(* Logix 5000 project; controller PLCbox vendor 1 type 14 code 149 rev 30.11; software revision 30.01 *)

TASK MainTask (continuous, watchdog 500 ms) : MainProgram, TestProgram, ExternalHardware, Riser, RPiEdgeIgnition, DellEdgeIgnition
TASK Projects (periodic, rate 10 ms, priority 10, watchdog 500 ms) : StreetLightSystem, PLC_Projects
TASK ST_Routines (periodic, rate 10 ms, priority 10, watchdog 500 ms) : ST_Practice
TASK Task100msec (periodic, rate 100 ms, priority 2, watchdog 500 ms) : MainProgram2
TASK Tutorials (periodic, rate 10 ms, priority 10, watchdog 500 ms) : Mathematical, InterviewPractice, CognexJobChange, Challenges_Projects, TankFillingChallenge, FTViewTutorial, Advanced, PowerFlex525Mastery, FIFOinstruction, JumpTest, DataTypes, PF525Control

MODULES
   Local : vendor 1 type 14 code 149 (Compact 0, rev 30.11)
      Discrete_IO : Embedded (Compact 1, rev 3.1, Output RPI 20 ms)
      CLX_PLC : 1756-EN2T (Ethernet 192.168.1.30, rev 5.28)
         CLX_MainPLC : vendor 1 type 14 code 54 (ICP 0, rev 20.4, $4ae8c327$ RPI 20 ms)
      PF1 : PowerFlex 525-EENET (Ethernet 192.168.1.7, rev 5.2, Output RPI 20 ms)
      Stratix1 : vendor 1 type 12 code 231 (Ethernet 192.168.1.10, rev 8.1, Output RPI 1000 ms)
      VladCognex : vendor 678 type 100 code 265 (Ethernet 192.168.1.15, rev 4.10, Output RPI 20 ms)
      Stratix2 : vendor 1 type 12 code 189 (Ethernet 192.168.1.12, rev 12.1, Output RPI 1000 ms)
      PointIORack1 : 1734-AENT (Ethernet 192.168.1.9, rev 5.1, Output RPI 20 ms)
         Local_IN2 : 1734-IB8 (PointIO 2, rev 3.1)
         Local_IN1 : 1734-IB8 (PointIO 1, rev 3.1)
         Local_OUT5 : vendor 1 type 7 code 288 (PointIO 5, rev 3.1)
         Local_OUT3 : 1734-OB8E (PointIO 3, rev 3.1)
         Local_IN4 : 1734-OA4 (PointIO 4, rev 3.1)
END_MODULES

TYPE String20 :
STRUCT
   LEN : DINT;
   DATA : SINT[20];
END_STRUCT
END_TYPE

TYPE UDT_BOOLarr :
STRUCT
   BOOLtag : BOOL[32];
END_STRUCT
END_TYPE

TYPE UDT_Output :
STRUCT
   Energize : BOOL;
   Auto : BOOL;
   ManualAvl : BOOL;
   Force : BOOL;
   ForceAvl : BOOL;
   Delay_ON : TIMER;
   Name : String20;
   SetAuto : BOOL;
   SetManual : BOOL;
   ForceON : BOOL;
   ForceOFF : BOOL;
END_STRUCT
END_TYPE

TYPE UDT_PID :
STRUCT
   P : REAL;
   I : REAL;
   D : REAL;
   CV : REAL;
   SP : REAL;
   PV : REAL;
   Auto : BOOL;
   Name : STRING;
END_STRUCT
END_TYPE

TYPE UDT_ProdCons :
STRUCT
   Status : CONNECTION_STATUS;
   Data : DINT[50];
END_STRUCT
END_TYPE

TYPE UDT_Time :
STRUCT
   Year : DINT;
   Month : DINT;
   Day : DINT;
   Hour : DINT;
   Minute : DINT;
   Second : DINT;
   Microsecond : DINT;
END_STRUCT
END_TYPE

TYPE UDT_VFD_PF525 :
STRUCT
   Start_PB : BOOL;
   Stop_PB : BOOL;
   Run : BOOL;
END_STRUCT
END_TYPE

TYPE Varchar40 :
STRUCT
   LEN : DINT;
   DATA : SINT[40];
END_STRUCT
END_TYPE

ADD_ON_INSTRUCTION AOI_BasicCalculation   (* revision 1.0, vendor SolisPLC *)
VAR_INPUT
   Operand_1 : REAL; {required}
   Operand_2 : REAL; {required}
   Operand_3 : REAL; {required}
   Operand_4 : REAL; {required}
END_VAR
VAR_OUTPUT
   Multiplication : REAL; {access Read Only, required}
   Addition : REAL; {access Read Only, required}
END_VAR
VAR
   Mul1 : REAL; {access None}
   Mul2 : REAL; {access None}
   Add1 : REAL; {access None}
   Add2 : REAL; {access None}
END_VAR

ROUTINE Logic   (* ladder *)
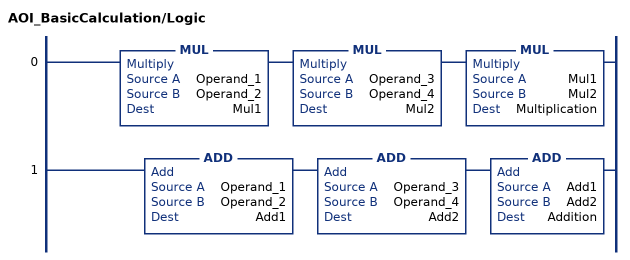
   0: MUL(Operand_1,Operand_2,Mul1)MUL(Operand_3,Operand_4,Mul2)MUL(Mul1,Mul2,Multiplication);
   1: ADD(Operand_1,Operand_2,Add1)ADD(Operand_3,Operand_4,Add2)ADD(Add1,Add2,Addition);
END_ROUTINE
END_ADD_ON_INSTRUCTION

ADD_ON_INSTRUCTION AOI_VFD_PF525   (* revision 1.0, vendor SolisPLC *)
VAR_IN_OUT
   VFD : UDT_VFD_PF525; {required}
END_VAR

ROUTINE Logic   (* structured text *)
   
END_ROUTINE
END_ADD_ON_INSTRUCTION

VAR_GLOBAL   (* controller tags *)
   AnalogInput : REAL[100] := ([0] := 5000.0);
   AnalogScaled : REAL[100] := ([0] := 93.75);
   ArrayOfBOOLs : DINT;
   BNOT_1501 : FBD_BOOLEAN_NOT := (In := 1);
   BOOL_IN_0 : BOOL;
   BOOL_OUT_0 : BOOL;
   BoxCounter : COUNTER := (PRE := 10, ACC := 10, DN := 1);
   Buttons : BOOL[64];
   Buttons2 : UDT_BOOLarr;
   Ch1_Volts : REAL;
   CLX_Cons : UDT_ProdCons := (Status.ConnectionFaulted := 1);
   CMPLX_Prod : UDT_ProdCons := (Status.RunMode := 1, Data[0] := 56789, Data[5] := 674); {produced}
   Command : BOOL[64];
   Condition : BOOL[32];
   Conv1Speed : REAL := 2.0;
   Conv2Speed_Fast : REAL := 3.0;
   Conv2Speed_Slow : REAL := 0.3;
   DINT_Arr1 : DINT[40] := ([0] := 1, [12] := 34534535, [31] := 131231, [34] := 123123);
   DINT_Arr2 : DINT[40] := ([0] := 1, [12] := 34534535, [31] := 131231);
   FaultedT : TIMER := (PRE := 2000, ACC := 860, EN := 1, TT := 1);
   FIFOControl3 : CONTROL := (LEN := 13, POS := 12);
   FIO_B_IN_0 : BOOL;   // Start Button
   FIO_B_IN_1 : BOOL := 1;   // Stop Button
   FIO_B_IN_2 : BOOL;   // System Running
   FIO_B_IN_3 : BOOL;   // Reset Button
   FIO_B_IN_4 : BOOL;
   FIO_B_IN_5 : BOOL;
   FIO_B_OUT_0 : BOOL;   // System Running - Confirmation
   FIO_B_OUT_1 : BOOL := 1;   // System Stopped - Confirmation
   FIO_B_OUT_2 : BOOL;   // System Faulted - Confirmation
   FIO_B_OUT_3 : BOOL := 1;   // Send boxes
   FIO_B_OUT_4 : BOOL := 1;
   FIO_B_OUT_5 : BOOL;
   FIO_B_OUT_6 : BOOL;
   FIO_F_OUT_0 : REAL;
   FIO_F_OUT_1 : REAL;
   FORDINT : DINT[30];
   FORDINT2 : DINT[30];
   HeatingSystem : REAL;
   HMI_Int_BOOL : BOOL[64] := ([5] := 1);
        [1]   // Light 1 Status - Yellow
        [2]   // Light 1 Status - Red
        [4]   // Light 2 Status - Yellow
        [5]   // Light 2 Status - Red
        [0]   // Light 1 Status - Green
        [3]   // Light 2 Status - Green
   HMI_Interface_BOOL : BOOL[64];
        [2]   // Light 1 - Red Status ON
        [5]   // Light 2 - Red Status ON
        [0]   // Light 1 - Green Status ON
        [1]   // Light 1 - Yellow Status ON
        [3]   // Light 2 - Green Status ON
        [4]   // Light 2 - Yellow Status ON
   HMI_No_Access : BOOL;
   IN_Loc1 : BOOL[32];
        [1]   // SPARE
        [2]   // SPARE
        [3]   // SPARE
        [4]   // SPARE
        [5]   // SPARE
        [6]   // SPARE
        [0]   // Box Counter P.E. - No Box
        [7]   // SPARE
   IN_Loc1_DB_OFF : BOOL[32];
   IN_Loc1_DB_ON : BOOL[32];
   IN_Loc1_Index : DINT := 7;
   IN_Loc1_T_OFF : TIMER[16] := ([0].PRE := 500, [0].ACC := 500);
   IN_Loc1_T_ON : TIMER[16] := ([0].PRE := 500);
   index : DINT := 50;
   JobData : SINT[32] := ([0] := 16, [2] := 70, [3] := 105, [4] := 114, [5] := 115, [6] := 116, [7] := 74, [8] := 111, [9] := 98, [10] := 84, [11] := 101, [12] := 115, [13] := 116, [14] := 46, [15] := 106, [16] := 111, [17] := 98);
   Light1_Complete_ONS : BOOL;
   Light1_Green : BOOL;
   Light1_Green_T : TIMER := (PRE := 10000);
   Light1_Red : BOOL;
   Light1_Reset : BOOL;
   Light1_Yellow : BOOL;
   Light1_Yellow_T : TIMER := (PRE := 3000);
   Light2_Complete_ONS : BOOL;
   Light2_Green : BOOL;
   Light2_Green_T : TIMER := (PRE := 10000);
   Light2_Red : BOOL;
   Light2_Reset : BOOL;
   Light2_Yellow : BOOL;
   Light2_Yellow_T : TIMER := (PRE := 3000);
   LightSystem_FLT : BOOL[64] := ([3] := 1);
        [1]   // FLT[1] - Light 1 - Yellow Light Faulted
        [0]   // FLT[0] - Light 1 - Green Light Faulted
   LightSystemFaulted : BOOL := 1;
   Local2IData : DINT := 53;
   Local3OData : DINT := 32;
   Local_IN_D : BOOL[256] := ([0] := 1, [2] := 1, [4] := 1, [5] := 1);
        [1]   // Light 1 - Yellow Light Corfirmed ON
        [0]   // Light 1 - Green Light Corfirmed ON
        [4]   // Light 2 - Yellow Light Corfirmed ON
        [2]   // Light 1 - Red Light Corfirmed ON
        [3]   // Light 2 - Green Light Corfirmed ON
        [5]   // Light 2 - Red Light Corfirmed ON
   Local_OUT_D : BOOL[256] := ([2] := 1);
        [0]   // Light 1 - Green Light Turn ON
        [2]   // Light 1 - Red Light Turn ON
        [3]   // Light 2 - Green Light Turn ON
        [1]   // Light 1 - Yellow Light Turn ON
        [5]   // Light 2 - Red Light Turn ON
        [4]   // Light 2 - Yellow Light Turn ON
   LocalOut : DINT[20] := ([2] := 548);
   LogicTag : BOOL[64] := ([12] := 1, [15] := 1);
   LoopDINT : DINT[30];
   LoopDINT2 : DINT[30];
   NewProductID : DINT := 1017;
   OUT_Loc1 : BOOL[32] := ([0] := 1);
   PID1 : PID := (CTL := 33920, INI := 1, DVNA := 1, PVHA := 1, SP := 200.0, KP := 1.0, KI := 0.1, KD := 0.1, MAXS := 1000.0, SO := 20.000076, MAXO := 100.0, UPD := 0.05, PV := 200.00174, ERR := -0.001739502, OUT := 20.000076, MAXI := 1000.0, MAXCV := 1000.0, MAXTIE := 100.0, DATA[0] := 20.00025, DATA[1] := -320.00278, DATA[2] := 200.00174, DATA[3] := -0.001739502, DATA[4] := 200.0, DATA[5] := 0.1, DATA[6] := 1.0, DATA[7] := 0.90000004, DATA[8] := 1.0, DATA[9] := 0.1, DATA[10] := 0.1, DATA[11] := 1.0, DATA[12] := 0.1, DATA[13] := 0.1, DATA[15] := 10.0, DATA[16] := 1.0);
   PID1_CV : REAL := 200.00076;
   PID1_PV : REAL := 200.00174;
   PID1_T : TIMER := (PRE := 50, ACC := 40, EN := 1, TT := 1);
   PID1_TB : REAL;
   PID_Analog_In : REAL[20];
   PID_Tutorial : PID := (CTL := 34432, INI := 1, DVNA := 1, DVPA := 1, PVHA := 1, SP := 100.0, KP := 5.0, KI := 5.0, KD := 5.0, MAXS := 1000.0, SO := 1.999996, MAXO := 100.0, UPD := 0.05, PV := 100.0, OUT := 1.999996, MAXI := 1000.0, MAXCV := 1000.0, MAXTIE := 100.0, DATA[0] := 1.9999565, DATA[1] := -160.00005, DATA[2] := 100.0, DATA[4] := 100.0, DATA[5] := 0.1, DATA[6] := 1.0, DATA[7] := 5.8, DATA[8] := 5.0, DATA[9] := 5.0, DATA[10] := 5.0, DATA[11] := 5.0, DATA[12] := 5.0, DATA[13] := 5.0, DATA[15] := 10.0, DATA[16] := 1.0);
   PLCTime : UDT_Time := (Year := 2020, Month := 4, Day := 20, Hour := 14, Minute := 9, Second := 30, Microsecond := 102344);
   Proj1_INT : INT[4] := ([0] := 16);
        [0].1   // System Faulted
        [0].2   // Enable Conveyor 1
        [0].3   // Enable Conveyor 2
        [0].4   // Conveyor 2 - HIGH SPEED
   RiserBOOL : BOOL[64];
        [7]   // Riser - Stop PB
        [8]   // Riser - Critical Fault
        [0]   // Riser - Cotnrol Valve OPEN
        [9]   // Riser - Fault Reset PB
        [5]   // Riser - Running Condition
        [4]   // Riser ALARM 004 - Pressure High High
        [3]   // Riser ALARM 003 - Pressure High
        [6]   // Riser - Start PB
        [2]   // Riser ALARM 002 - Pressure Low
        [1]   // Riser ALARM 001 - Pressure Low Low
   RiserREAL : REAL[20] := ([0] := 55.0, [1] := 20.0, [2] := 5.0, [3] := 124.80001, [4] := 140.40001, [5] := 140.0, [6] := 156.00002, [7] := 124.80001, [8] := 140.40001, [9] := 4.0, [10] := 4.5);
        [1]   // Riser - Pressure Limit Low Low[PSI]
        [2]   // Riser - Pressure Limit Low [PSI]
        [0]   // Riser - Current Pressure Reading [PSI]
        [6]   // Riser - DR 9 Pipe Pressure Rating [PSI]
        [5]   // Riser - Current Temperature Reading [deg F]
        [4]   // Riser - Pressure Limit High High [PSI]
        [3]   // Riser - Pressure Limit High [PSI]
        [8]   // Riser - Pressure Limit High High [PSI]
        [7]   // Riser - Pressure Limit High [PSI]
   SCLA_10 : SCALE := (In := 5000.0, InRawMax := 16000.0, InEUMax := 300.0, Out := 93.75);
   SCLA_11 : SCALE;
   SCLA_12 : SCALE;
   SetJob : MESSAGE;
        MessageParameters(ServiceCode := 16#0010, LocalElement := JobData[0], ...)
   SolisBOOL : BOOL[64] := ([2] := 1, [3] := 1, [4] := 1, [5] := 1, [7] := 1, [8] := 1, [9] := 1, [10] := 1, [11] := 1, [12] := 1, [13] := 1);
   SolisDINT : DINT[20] := ([2] := 42, [3] := 234, [5] := 234, [6] := 33, [7] := 234, [8] := 234, [9] := 23, [10] := 24, [11] := 42, [12] := 234, [13] := 423, [15] := 42);
   SolisREAL : REAL[20];
   SsytemStopped : BOOL := 1;
   StatusInt : DINT := 2;
   System_Timer : TIMER[100] := ([0].PRE := 10000, [0].ACC := 783, [0].EN := 1, [0].TT := 1);
   SystemFaultReset : BOOL;
   tagToPi : DINT := 119;
   TempSensor : REAL;
   TIC_1501 : PID_ENHANCED := (PVEUMax := 100.0, SPHLimit := 100.0, RatioProg := 1.0, RatioOper := 1.0, RatioHLimit := 1.0, RatioLLimit := 1.0, CVEUMax := 100.0, CVHLimit := 100.0, PVEDerivative := 1, RTSTime := 1);
END_VAR

PROGRAM Advanced   (* main routine _01_Main *)
VAR
   Add : REAL;
   AOI_Basic1 : AOI_BasicCalculation;
   Array1_INT : INT[10] := ([0] := -21846, [1] := -1);
   Array2_DINT : DINT[10] := ([0] := -21846);
   BatchCompletedConfirm : BOOL;
   Data : DINT[50];
   Data2 : DINT[50];
   DestBit : DINT;
   Ingredient1Stp : DINT := 30;
   Ingredient2Stp : DINT := 70;
   Ingredient3Stp : DINT := 99;
   Mult : REAL;
   Op1 : REAL;
   Op2 : REAL;
   Op3 : REAL;
   Op4 : REAL;
   PLCCond : BOOL[32];
        [1]   // Batch Start Button
   PLCCondOut : BOOL[32] := ([1] := 1);
        [8]   // Batch Completed
        [2]   // Ingredient 1 Valve OPEN
        [1]   // Tank Ready for Batch
        [4]   // Enable Stirrer (VFD)
        [5]   // Hops Feeder ENABLE
        [3]   // Ingredient 2 Valve OPEN
        [6]   // Tank Heating System ENABLE
   SeqArr : DINT[10] := ([0] := 1, [1] := 2, [2] := 4, [3] := 12, [4] := 28, [5] := 60, [6] := 124, [7] := 128);
   SeqArr2 : DINT[10] := ([0] := 1, [1] := 2, [2] := 4, [3] := 24, [4] := 48, [5] := 80, [6] := 208, [7] := 256);
   SeqControl : CONTROL := (LEN := 7, POS := 1);
   SeqMask : DINT := 65535;
   SeqOut : DINT := 2;
   SeqSource : DINT;
   SequencePosition : DINT;
   SequenceStart : BOOL;
   SrcBit : DINT;
   TankDelay : TIMER := (PRE := 30000);
   TankLevel : DINT;
   TankTemperature : DINT := 200;
   TankTempStp : DINT := 220;
END_VAR

ROUTINE _01_Main   (* ladder *)
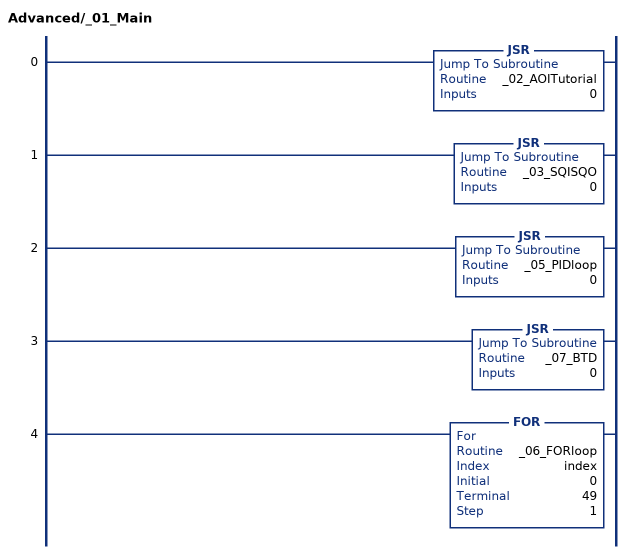
   0: JSR(_02_AOITutorial,0);
   1: JSR(_03_SQISQO,0);
   2: JSR(_05_PIDloop,0);
   3: JSR(_07_BTD,0);
   4: FOR(_06_FORloop,index,0,49,1);
END_ROUTINE

ROUTINE _02_AOITutorial   (* ladder *)
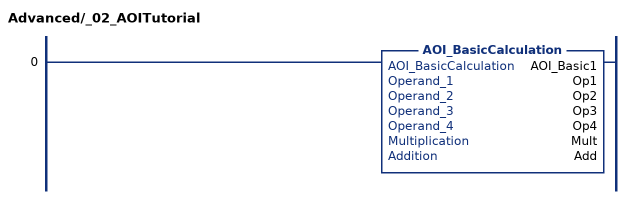
   0: AOI_BasicCalculation(AOI_Basic1,Op1,Op2,Op3,Op4,Mult,Add);
END_ROUTINE

ROUTINE _03_SQISQO   (* ladder *)
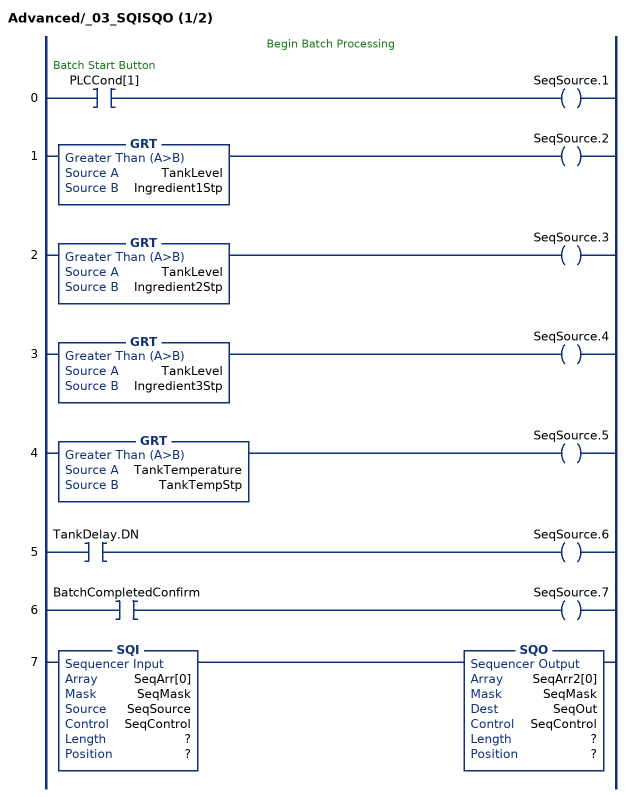
   // Begin Batch Processing
   0: XIC(PLCCond[1])OTE(SeqSource.1);
   1: GRT(TankLevel,Ingredient1Stp)OTE(SeqSource.2);
   2: GRT(TankLevel,Ingredient2Stp)OTE(SeqSource.3);
   3: GRT(TankLevel,Ingredient3Stp)OTE(SeqSource.4);
   4: GRT(TankTemperature,TankTempStp)OTE(SeqSource.5);
   5: XIC(TankDelay.DN)OTE(SeqSource.6);
   6: XIC(BatchCompletedConfirm)OTE(SeqSource.7);
   7: SQI(SeqArr[0],SeqMask,SeqSource,SeqControl,?,?)SQO(SeqArr2[0],SeqMask,SeqOut,SeqControl,?,?);
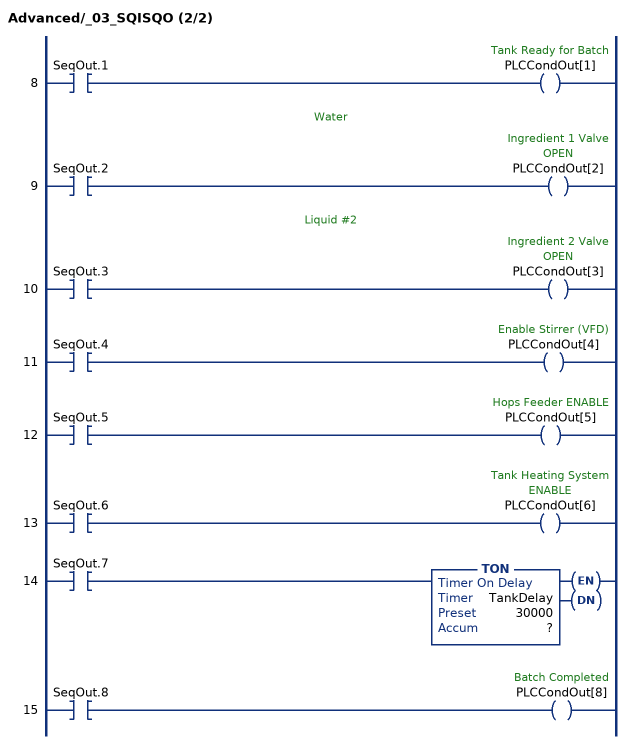
   8: XIC(SeqOut.1)OTE(PLCCondOut[1]);
   // Water
   9: XIC(SeqOut.2)OTE(PLCCondOut[2]);
   // Liquid #2
   10: XIC(SeqOut.3)OTE(PLCCondOut[3]);
   11: XIC(SeqOut.4)OTE(PLCCondOut[4]);
   12: XIC(SeqOut.5)OTE(PLCCondOut[5]);
   13: XIC(SeqOut.6)OTE(PLCCondOut[6]);
   14: XIC(SeqOut.7)TON(TankDelay,?,?);
   15: XIC(SeqOut.8)OTE(PLCCondOut[8]);
END_ROUTINE

ROUTINE _05_PIDloop   (* ladder *)
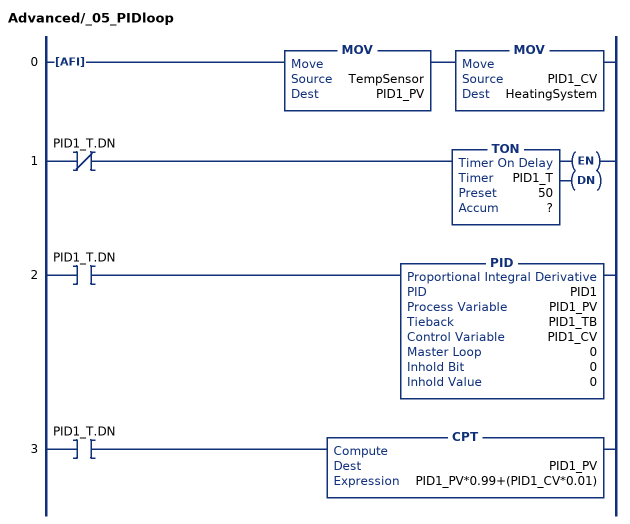
   0: AFI()MOV(TempSensor,PID1_PV)MOV(PID1_CV,HeatingSystem);
   1: XIO(PID1_T.DN)TON(PID1_T,?,?);
   2: XIC(PID1_T.DN)PID(PID1,PID1_PV,PID1_TB,PID1_CV,0,0,0);
   3: XIC(PID1_T.DN)CPT(PID1_PV,PID1_PV*0.99+(PID1_CV*0.01));
END_ROUTINE

ROUTINE _06_FORloop   (* ladder *)
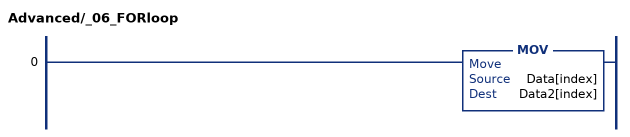
   0: MOV(Data[index],Data2[index]);
END_ROUTINE

ROUTINE _07_BTD   (* ladder *)
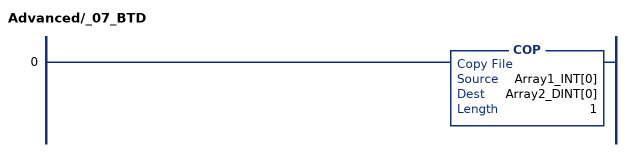
   0: COP(Array1_INT[0],Array2_DINT[0],1);
END_ROUTINE
END_PROGRAM

PROGRAM Challenges_Projects   (* main routine _01_Main *)
VAR
   GREEN_LIGHT_ON : BOOL;
   RED_LIGHT_ON : BOOL;
   RESET_PRESSED : BOOL;
   START_PRESSED : BOOL;
   STOP_PRESSED : BOOL;
   YELLOW_LIGHT_ON : BOOL;
END_VAR

ROUTINE _01_Main   (* ladder *)
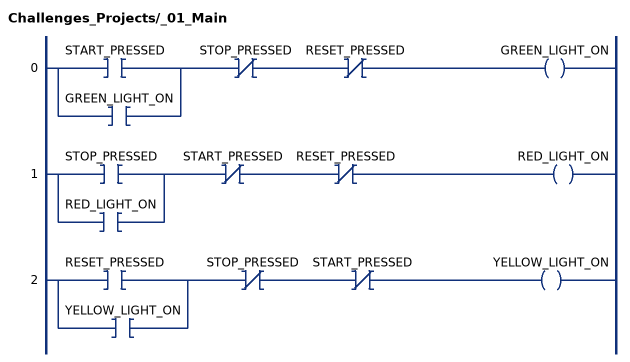
   0: [XIC(START_PRESSED) ,XIC(GREEN_LIGHT_ON) ]XIO(STOP_PRESSED)XIO(RESET_PRESSED)OTE(GREEN_LIGHT_ON);
   1: [XIC(STOP_PRESSED) ,XIC(RED_LIGHT_ON) ]XIO(START_PRESSED)XIO(RESET_PRESSED)OTE(RED_LIGHT_ON);
   2: [XIC(RESET_PRESSED) ,XIC(YELLOW_LIGHT_ON) ]XIO(STOP_PRESSED)XIO(START_PRESSED)OTE(YELLOW_LIGHT_ON);
END_ROUTINE
END_PROGRAM

PROGRAM CognexJobChange   (* main routine Main *)
VAR
   JobIndex : DINT := 1;
   JobName : STRING[10] := ([0] := 'VladsJob.job', [1] := 'FirstJobTest.job', [2] := 'BarcodeRead.job');
   JobSet : BOOL[32];
   JobTrigger : BOOL;
   TriggerONS : BOOL;
   VladsCounter : COUNTER := (ACC := 11, DN := 1);
END_VAR

ROUTINE Main   (* ladder *)
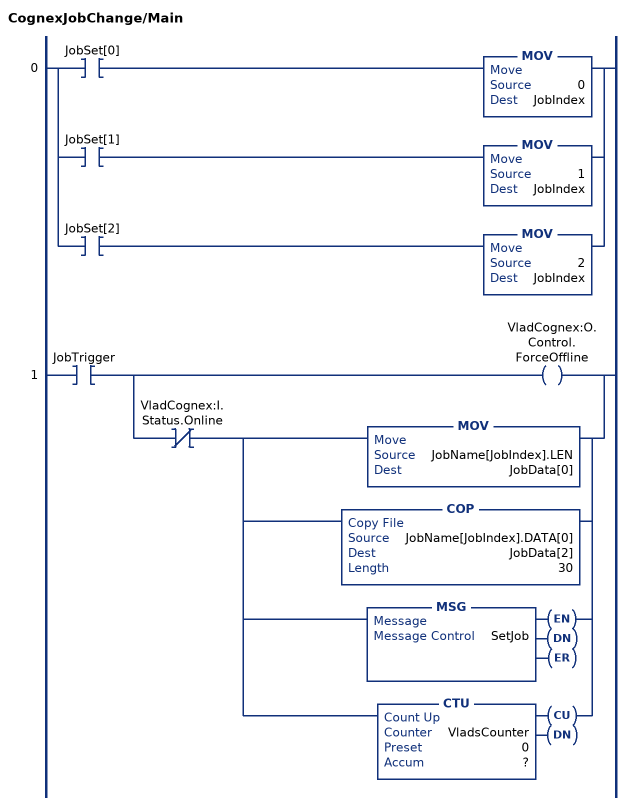
   0: [XIC(JobSet[0]) MOV(0,JobIndex) ,XIC(JobSet[1]) MOV(1,JobIndex) ,XIC(JobSet[2]) MOV(2,JobIndex) ];
   1: XIC(JobTrigger)[OTE(VladCognex:O.Control.ForceOffline) ,XIO(VladCognex:I.Status.Online) [MOV(JobName[JobIndex].LEN,JobData[0]) ,COP(JobName[JobIndex].DATA[0],JobData[2],30) ,MSG(SetJob) ,CTU(VladsCounter,?,?) ] ];
END_ROUTINE
END_PROGRAM

PROGRAM DataTypes   (* main routine _01_Main *)
VAR
   Machine : BOOL := 1;
   Output : DINT := 7;
   Output2 : DINT := 7;
   Output_Buffer1 : DINT := 7;
   Start_Light : BOOL := 1;
   Stop_Light : BOOL := 1;
   Tag1 : BOOL := 1;
   Tag10 : DINT[10] := ([5] := 256);
   Tag2 : INT;
   Tag3 : DINT;
   Tag4 : BOOL[32] := ([2] := 1, [5] := 1, [8] := 1, [11] := 1, [17] := 1);
   Tag5 : DINT;
   Tag6 : BOOL;
   Tag7 : BOOL;
   Tag8 : DINT;
   Tag9 : BOOL;
   ValveOutput : BOOL := 1;
   Warning_Light : BOOL := 1;
END_VAR

ROUTINE _01_Main   (* ladder *)
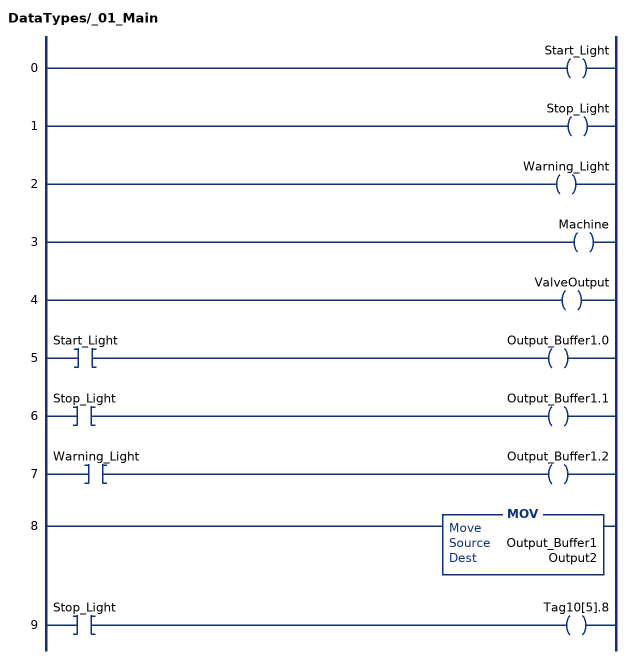
   0: OTE(Start_Light);
   1: OTE(Stop_Light);
   2: OTE(Warning_Light);
   3: OTE(Machine);
   4: OTE(ValveOutput);
   5: XIC(Start_Light)OTE(Output_Buffer1.0);
   6: XIC(Stop_Light)OTE(Output_Buffer1.1);
   7: XIC(Warning_Light)OTE(Output_Buffer1.2);
   8: MOV(Output_Buffer1,Output2);
   9: XIC(Stop_Light)OTE(Tag10[5].8);
END_ROUTINE
END_PROGRAM

PROGRAM DellEdgeIgnition
VAR
   DellIgn_BOOL : BOOL[128];
   DellIgn_DINT : DINT[50] := ([0] := 1);
END_VAR
END_PROGRAM

PROGRAM ExternalHardware   (* main routine _01_Main *)
VAR
   HMI_O_Screeen_Title : String20[100] := ([0] := 'Slot 0 - Local Out.', [1] := 'Main Screen', [2] := 'System Settings', [3] := 'In Q - Motor Starter', [4] := 'Alarm Display');
END_VAR

ROUTINE _01_Main   (* ladder *)
   0 (stored rung type 13): ;
END_ROUTINE
END_PROGRAM

PROGRAM FIFOinstruction   (* main routine FIFOdemo *)
VAR
   BoxCounter2 : COUNTER := (ACC := 1, CU := 1, DN := 1);
   BoxProx2 : BOOL := 1;
   FIFO_Array : DINT[100] := ([0] := 140, [1] := 12910, [2] := 440, [3] := 150, [4] := 150, [5] := 150, [6] := 180, [7] := 300, [8] := 109, [9] := 10, [10] := 130, [11] := 180, [12] := 160, [13] := 240, [14] := 780, [15] := 880, [16] := 300000, [17] := 250, [18] := 150);
   FIFO_Array3 : DINT[100] := ([0] := 1, [1] := 1, [2] := 1, [3] := 1, [4] := 1, [5] := 1, [6] := 1, [7] := 1, [8] := 1, [9] := 1, [10] := 1, [11] := 1);
   FIFO_Unld : DINT := 1;
   FIFOAvg : DINT := 1;
   FIFOControl : CONTROL := (LEN := 20, POS := 19);
   FIFOLength : DINT := 11;
   FIFOSum : DINT := 12;
   SecTime : DINT;
   System_BOOL : BOOL;
   System_BOOL1 : BOOL[64] := ([5] := 1);
   TimerSinceLastBox : TIMER := (PRE := 300000, ACC := 300000, EN := 1, DN := 1);
END_VAR

ROUTINE FIFO_Avg   (* ladder *)
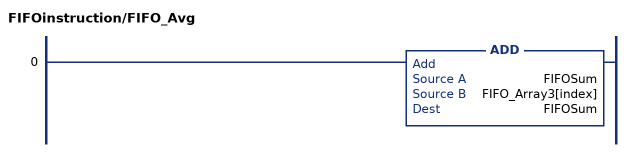
   0: ADD(FIFOSum,FIFO_Array3[index],FIFOSum);
END_ROUTINE

ROUTINE FIFOdemo   (* ladder *)
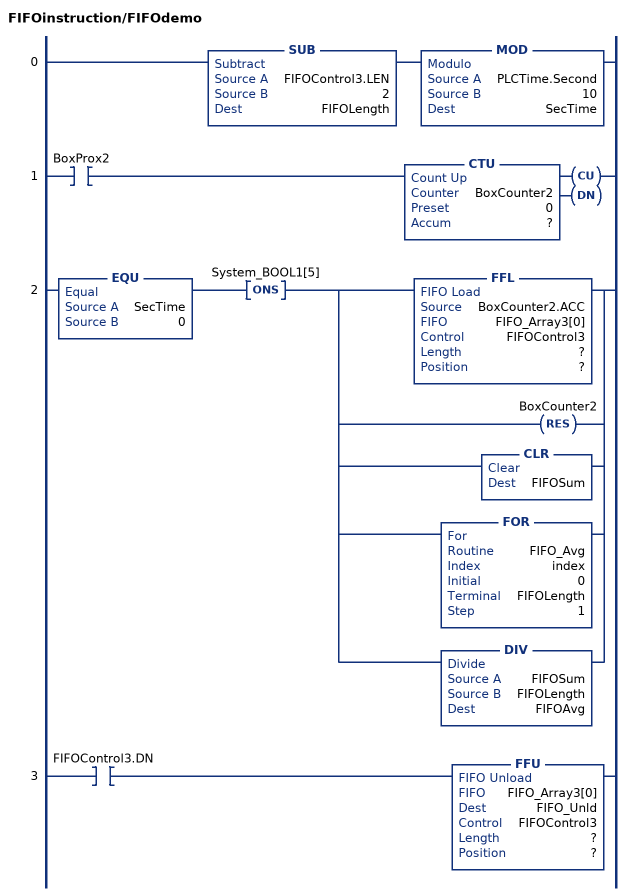
   0: SUB(FIFOControl3.LEN,2,FIFOLength)MOD(PLCTime.Second,10,SecTime);
   1: XIC(BoxProx2)CTU(BoxCounter2,?,?);
   2: EQU(SecTime,0)ONS(System_BOOL1[5])[FFL(BoxCounter2.ACC,FIFO_Array3[0],FIFOControl3,?,?) ,RES(BoxCounter2) ,CLR(FIFOSum) ,FOR(FIFO_Avg,index,0,FIFOLength,1) ,DIV(FIFOSum,FIFOLength,FIFOAvg) ];
   3: XIC(FIFOControl3.DN)FFU(FIFO_Array3[0],FIFO_Unld,FIFOControl3,?,?);
END_ROUTINE
END_PROGRAM

PROGRAM FTViewTutorial   (* main routine _01_Main *)
VAR
   AlarmReset : BOOL;
   HMI_Rotation : TIMER := (PRE := 5000, ACC := 410, EN := 1, TT := 1);
   HMI_Rotation_Enable : BOOL := 1;
   Motor1HL : BOOL;
   Motor1LL : BOOL;
   Motor1Speed : REAL := 60.0;
   Motor1SpeedActual : REAL := 60.0;
   Motor1SpeedSetpoint : REAL := 60.0;
   Motor1Var : REAL := 5.0;
END_VAR

ROUTINE _01_Main   (* ladder *)
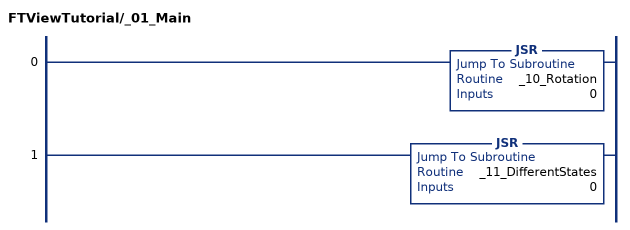
   0: JSR(_10_Rotation,0);
   1: JSR(_11_DifferentStates,0);
END_ROUTINE

ROUTINE _10_Rotation   (* ladder *)
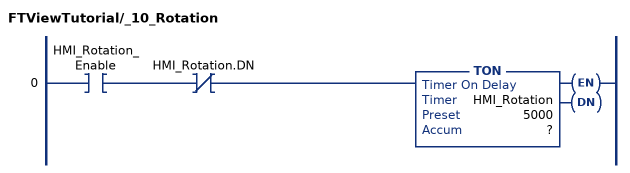
   0: XIC(HMI_Rotation_Enable)XIO(HMI_Rotation.DN)TON(HMI_Rotation,?,?);
END_ROUTINE

ROUTINE _11_DifferentStates   (* ladder *)
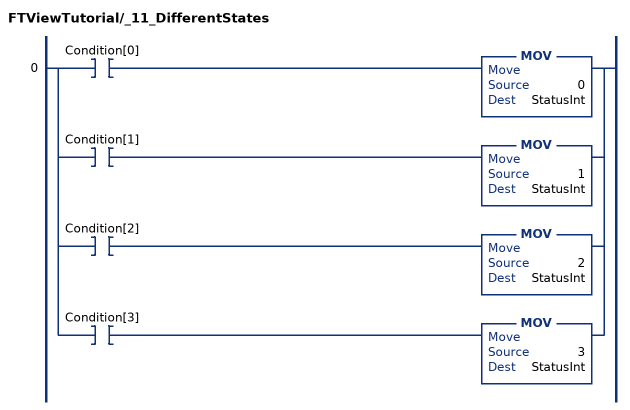
   0: [XIC(Condition[0]) MOV(0,StatusInt) ,XIC(Condition[1]) MOV(1,StatusInt) ,XIC(Condition[2]) MOV(2,StatusInt) ,XIC(Condition[3]) MOV(3,StatusInt) ];
END_ROUTINE
END_PROGRAM

PROGRAM InterviewPractice   (* main routine _01_Main *)
VAR
   AllOn : DINT := 2;
   CurrentRecipe : DINT := 2;
   HMI_RecipeSelected : DINT := 2;
   INT_Motor : BOOL[32];
        [1]   // STOP
        [10]   // MOTOR STARTER
        [0]   // START
        [2]   // MOTOR OVERLOAD / FAULT
   Recipe : DINT[10] := ([0] := 255, [1] := 55);
   RecipeCheck : DINT[10] := ([1] := 55);
   RecipeChk : DINT[10] := ([1] := 55, [2] := 10, [3] := 48);
   RecipeNumber : DINT[10] := ([1] := 55, [2] := 10, [3] := 48);
   SensorValve : DINT := 11;
   test : BOOL := 1;
   ValveBank : BOOL[32];
        [0]   // Valve - Sugar Tank
        [1]   // Valve - Salt Tank
        [2]   // Valve - Spice Tank
        [3]   // Valve - Iodine Tank
   ValveBank2 : BOOL[32] := ([0] := 1, [1] := 1, [2] := 1, [3] := 1, [4] := 1, [5] := 1, [6] := 1);
   ValveBank3 : DINT := 2;
   ValveBits : DINT;
   Valves : DINT := 10;
        .1   // Ingredient Valve - Salt
        .2   // Ingredient Valve - Spices
        .0   // Ingredient Valve - Sugar
        .3   // Ingredient Valve - Malto
   ValvesOK_SystemReady : BOOL;
   ValvesOK_SystemReady2 : BOOL := 1;
   ValvesOpen : DINT := 11;
END_VAR

ROUTINE _01_Main   (* ladder *)
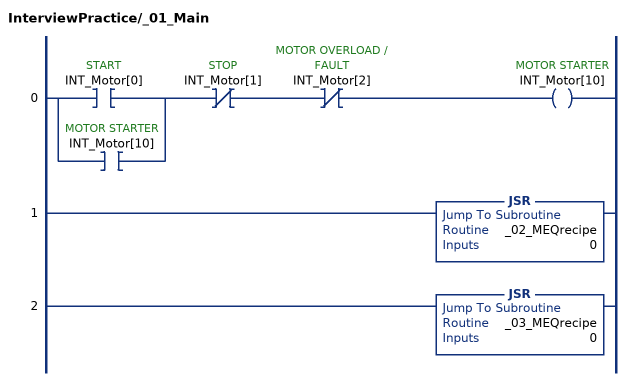
   0: [XIC(INT_Motor[0]) ,XIC(INT_Motor[10]) ]XIO(INT_Motor[1])XIO(INT_Motor[2])OTE(INT_Motor[10]);
   1: JSR(_02_MEQrecipe,0);
   2: JSR(_03_MEQrecipe,0);
END_ROUTINE

ROUTINE _02_MEQrecipe   (* ladder *)
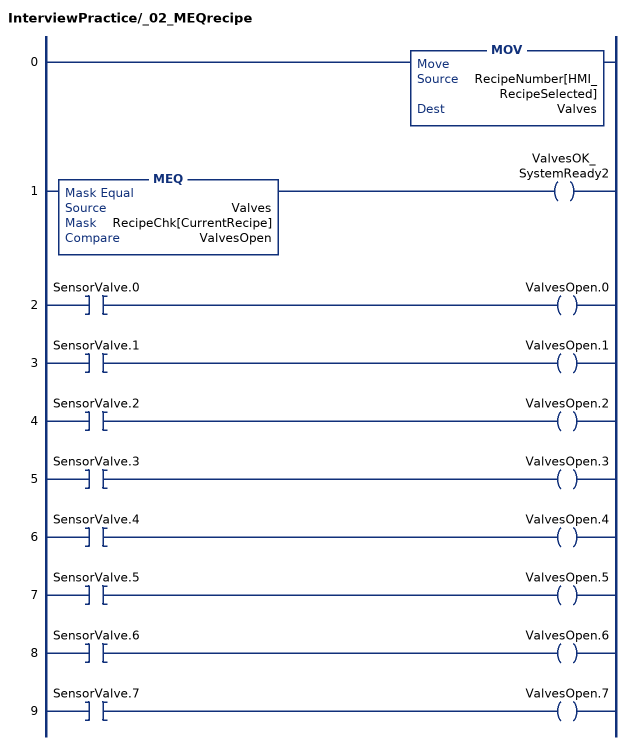
   0: MOV(RecipeNumber[HMI_RecipeSelected],Valves);
   1: MEQ(Valves,RecipeChk[CurrentRecipe],ValvesOpen)OTE(ValvesOK_SystemReady2);
   2: XIC(SensorValve.0)OTE(ValvesOpen.0);
   3: XIC(SensorValve.1)OTE(ValvesOpen.1);
   4: XIC(SensorValve.2)OTE(ValvesOpen.2);
   5: XIC(SensorValve.3)OTE(ValvesOpen.3);
   6: XIC(SensorValve.4)OTE(ValvesOpen.4);
   7: XIC(SensorValve.5)OTE(ValvesOpen.5);
   8: XIC(SensorValve.6)OTE(ValvesOpen.6);
   9: XIC(SensorValve.7)OTE(ValvesOpen.7);
END_ROUTINE
